// TIA Portal V19 export
FUNCTION_BLOCK "HMIGraphicControl"   // FB4, LAD
{ S7_Optimized_Access := 'TRUE' }
// stored: MemoryReserve 100, SetENOAutomatically false
   VAR_INPUT
      "Conveyor Speed" { ExternalAccessible := 'False'; ExternalVisible := 'False'; ExternalWritable := 'False'} : Real;   // m/min
      "Arm Speed" { ExternalAccessible := 'False'; ExternalVisible := 'False'; ExternalWritable := 'False'} : Real;   // m/min
      "Conveyor Max Speed" { ExternalAccessible := 'False'; ExternalVisible := 'False'; ExternalWritable := 'False'} : Real := 3000.0;
      "Arm Max Speed" { ExternalAccessible := 'False'; ExternalVisible := 'False'; ExternalWritable := 'False'} : Real := 32000.0;
      ConveyorMoving : Bool := true;
      ArmMoving : Bool := true;
      Reset : Bool;
   END_VAR
   VAR_OUTPUT
      Conveyor_On : Bool;
      Arm_On : Bool;
   END_VAR
   VAR_IN_OUT
      System_Enable : Bool;
      Graphic_Index { ExternalAccessible := 'False'; ExternalVisible := 'False'; ExternalWritable := 'False'} : Int;
      Box_Cnt : DInt;
      Pallet_Cnt : DInt;
   END_VAR
   VAR
      IEC_Timer_0_Instance { S7_SetPoint := 'True'} : IEC_TIMER;
      ConveyorTick : Bool;
      ConveyorTime : DInt;
      ConveyorTimeFactor : DInt := 100000;
      ArmTick : Bool;
      ArmTimeFactor : DInt := 100000;
      ArmTime : DInt;
      IEC_Timer_0_Instance_1 { S7_SetPoint := 'True'} : IEC_TIMER;
   END_VAR
   VAR_TEMP
      ConveyorScaled : Real;
      ConveyMotor : Bool;
      ArmScaled : Real;
   END_VAR
   VAR_TEMP   // added for the SCL form of the ladder/FBD networks
      _w1 : Bool;
   END_VAR
BEGIN

REGION Network 1
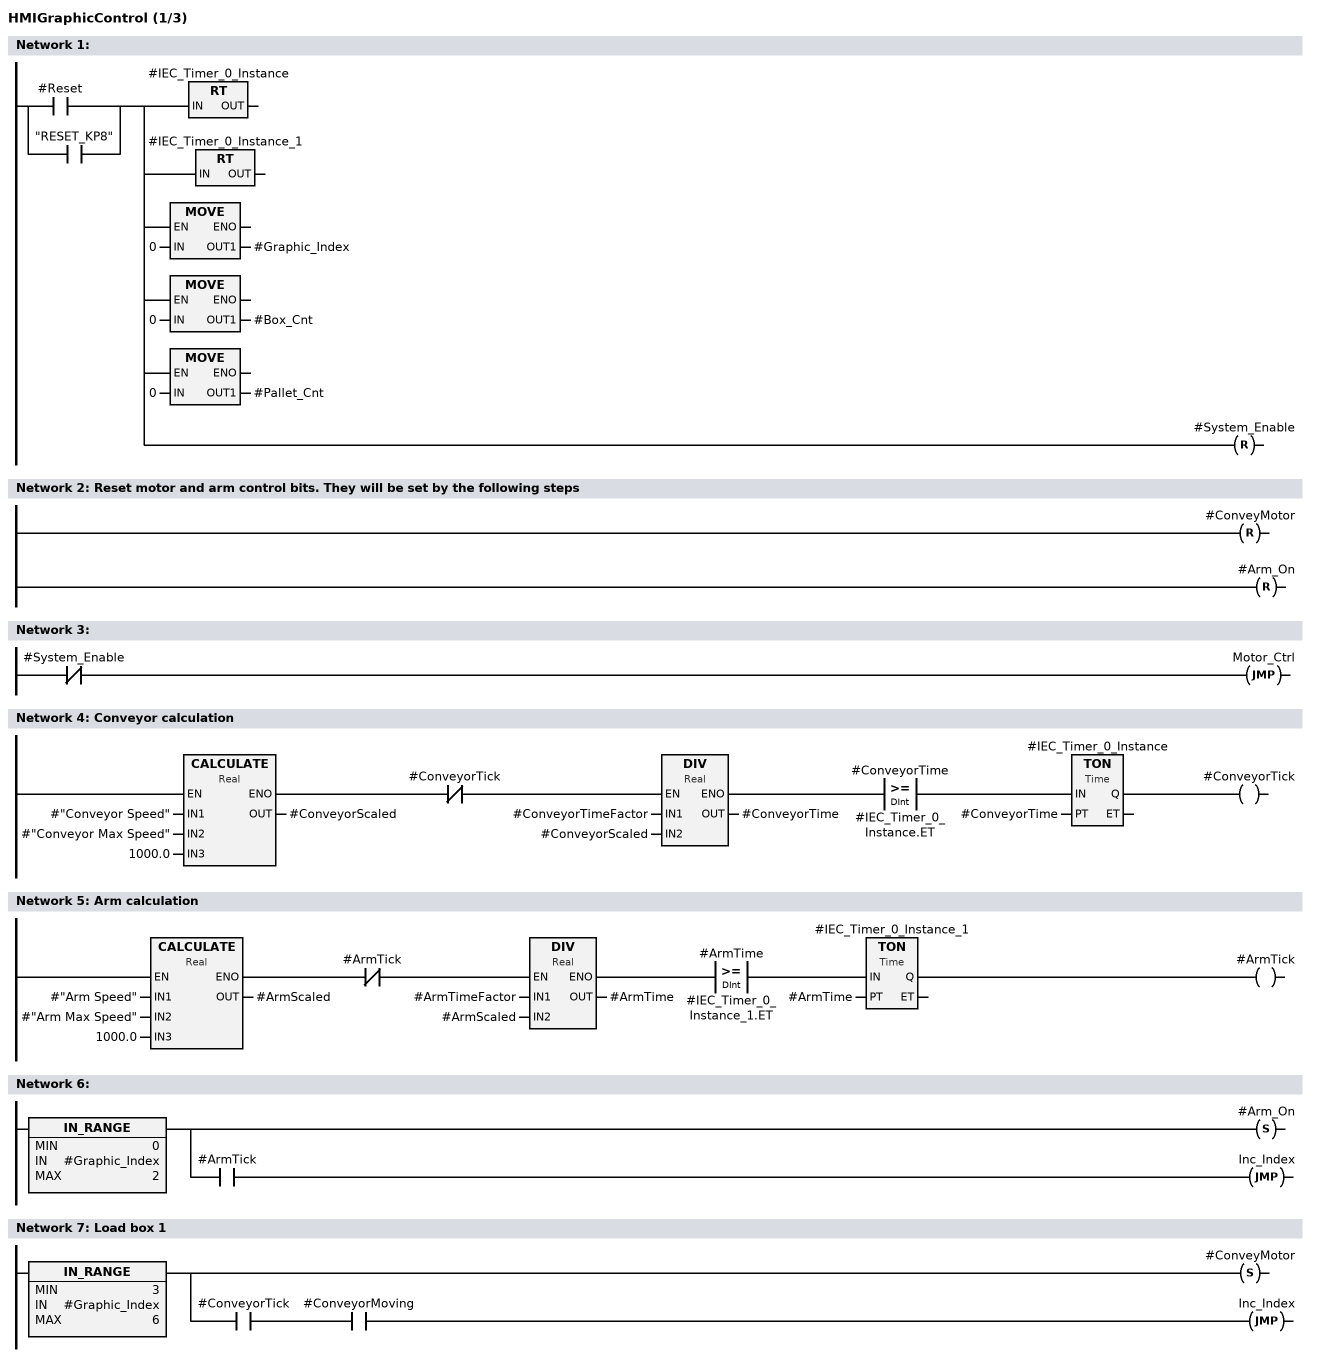
   RUNG wire#powerrail
      Contact( #Reset )
      wire#w1
      RT_Coil( #IEC_Timer_0_Instance )
   END_RUNG
   RUNG wire#powerrail
      Contact( "RESET_KP8" )
   END_RUNG wire#w1
   RUNG wire#w1
      RT_Coil( #IEC_Timer_0_Instance_1 )
   END_RUNG
   RUNG wire#w1
      Move(in := 0, out1 => #Graphic_Index)
   END_RUNG
   RUNG wire#w1
      Move(in := 0, out1 => #Box_Cnt)
   END_RUNG
   RUNG wire#w1
      Move(in := 0, out1 => #Pallet_Cnt)
   END_RUNG
   RUNG wire#w1
      R_Coil( #System_Enable )
   END_RUNG
   // the same network as SCL:
   #_w1 := #Reset OR "RESET_KP8";
   IF #_w1 THEN
       RESET_TIMER(#IEC_Timer_0_Instance);
       RESET_TIMER(#IEC_Timer_0_Instance_1);
       #Graphic_Index := 0;
       #Box_Cnt := 0;
       #Pallet_Cnt := 0;
       #System_Enable := FALSE;
   END_IF;
END_REGION

REGION Network 2: Reset motor and arm control bits. They will be set by the following steps
   RUNG wire#powerrail
      R_Coil( #ConveyMotor )
   END_RUNG
   RUNG wire#powerrail
      R_Coil( #Arm_On )
   END_RUNG
   // the same network as SCL:
   #ConveyMotor := FALSE;
   #Arm_On := FALSE;
END_REGION

REGION Network 3
   RUNG wire#powerrail
      I_Contact( #System_Enable )
      JumpCoil( Motor_Ctrl )
   END_RUNG
   // the same network as SCL:
   IF NOT #System_Enable THEN GOTO Motor_Ctrl; END_IF;
END_REGION

REGION Network 4: Conveyor calculation
   RUNG wire#powerrail
      { S7_Templates := "SrcType := Real"; S7_Expression := "IN1/IN2*IN3" } Calculate(in1 := #"Conveyor Speed", in2 := #"Conveyor Max Speed", in3 := 1000.0, out => #ConveyorScaled)
      I_Contact( #ConveyorTick )
      { S7_Templates := "SrcType := Real"; S7_GenerateENO := "TRUE" } Div(in1 := #ConveyorTimeFactor, in2 := #ConveyorScaled, out => #ConveyorTime)
      { S7_Templates := "SrcType := DInt" } GE_Contact(in1 := #ConveyorTime, in2 := #IEC_Timer_0_Instance.ET)
      { S7_Templates := "time_type := Time" } #IEC_Timer_0_Instance.TON(pt := #ConveyorTime, et =>)
      Coil( #ConveyorTick )
   END_RUNG
   // the same network as SCL:
   // ENO of a box is taken as its EN; it also drops when the box reports an error
   #ConveyorScaled := #"Conveyor Speed"/#"Conveyor Max Speed"*1000.0;
   IF NOT #ConveyorTick THEN #ConveyorTime := #ConveyorTimeFactor / #ConveyorScaled; END_IF;
   #IEC_Timer_0_Instance.TON(IN := NOT #ConveyorTick AND (#ConveyorTime >= #IEC_Timer_0_Instance.ET),
                           PT := #ConveyorTime);
   #ConveyorTick := #IEC_Timer_0_Instance.Q;
END_REGION

REGION Network 5: Arm calculation
   RUNG wire#powerrail
      { S7_Templates := "SrcType := Real"; S7_Expression := "IN1/IN2*IN3" } Calculate(in1 := #"Arm Speed", in2 := #"Arm Max Speed", in3 := 1000.0, out => #ArmScaled)
      I_Contact( #ArmTick )
      { S7_Templates := "SrcType := Real"; S7_GenerateENO := "TRUE" } Div(in1 := #ArmTimeFactor, in2 := #ArmScaled, out => #ArmTime)
      { S7_Templates := "SrcType := DInt" } GE_Contact(in1 := #ArmTime, in2 := #IEC_Timer_0_Instance_1.ET)
      { S7_Templates := "time_type := Time" } #IEC_Timer_0_Instance_1.TON(pt := #ArmTime, et =>)
      Coil( #ArmTick )
   END_RUNG
   // the same network as SCL:
   // ENO of a box is taken as its EN; it also drops when the box reports an error
   #ArmScaled := #"Arm Speed"/#"Arm Max Speed"*1000.0;
   IF NOT #ArmTick THEN #ArmTime := #ArmTimeFactor / #ArmScaled; END_IF;
   #IEC_Timer_0_Instance_1.TON(IN := NOT #ArmTick AND (#ArmTime >= #IEC_Timer_0_Instance_1.ET), PT := #ArmTime);
   #ArmTick := #IEC_Timer_0_Instance_1.Q;
END_REGION

REGION Network 6
   RUNG wire#powerrail
      { S7_Templates := "SrcType := Int" } InRange(min := 0, in := #Graphic_Index, max := 2)
      wire#w1
      S_Coil( #Arm_On )
   END_RUNG
   RUNG wire#w1
      Contact( #ArmTick )
      JumpCoil( Inc_Index )
   END_RUNG
   // the same network as SCL:
   #_w1 := (0 <= #Graphic_Index) AND (#Graphic_Index <= 2);
   IF #_w1 THEN #Arm_On := TRUE; END_IF;
   IF #_w1 AND #ArmTick THEN GOTO Inc_Index; END_IF;
END_REGION

REGION Network 7: Load box 1
   RUNG wire#powerrail
      { S7_Templates := "SrcType := Int" } InRange(min := 3, in := #Graphic_Index, max := 6)
      wire#w1
      S_Coil( #ConveyMotor )
   END_RUNG
   RUNG wire#w1
      Contact( #ConveyorTick )
      Contact( #ConveyorMoving )
      JumpCoil( Inc_Index )
   END_RUNG
   // the same network as SCL:
   #_w1 := (3 <= #Graphic_Index) AND (#Graphic_Index <= 6);
   IF #_w1 THEN #ConveyMotor := TRUE; END_IF;
   IF #_w1 AND #ConveyorTick AND #ConveyorMoving THEN GOTO Inc_Index; END_IF;
END_REGION

REGION Network 8
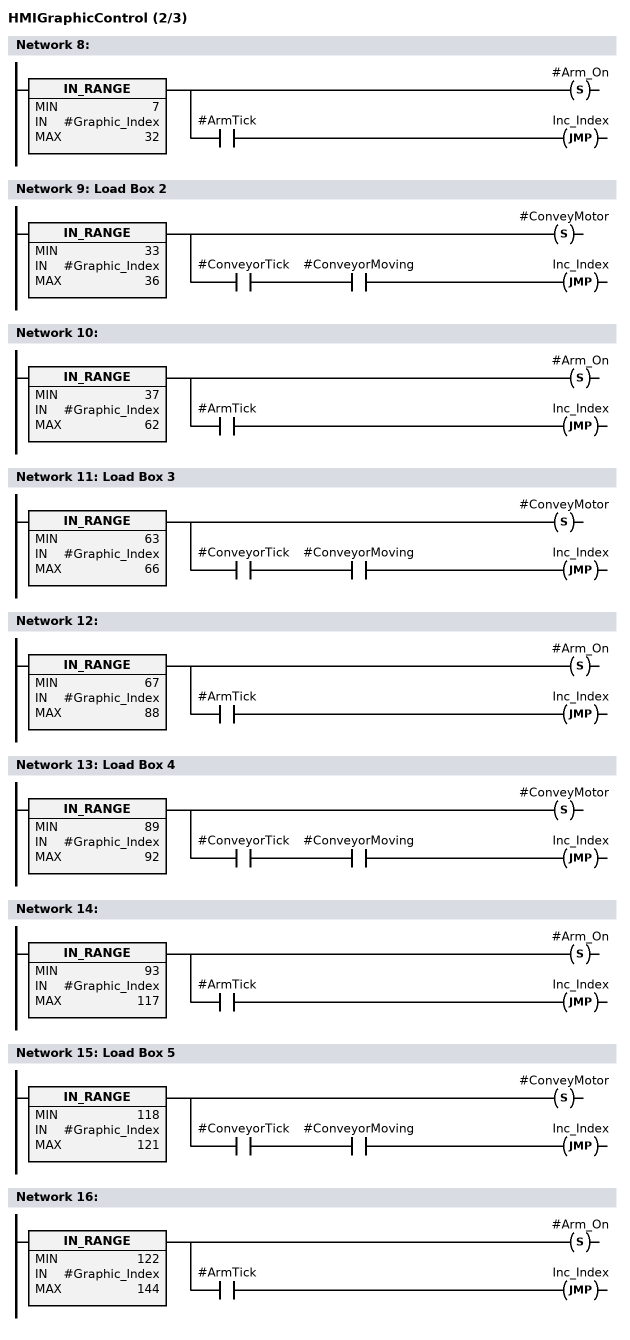
   RUNG wire#powerrail
      { S7_Templates := "SrcType := Int" } InRange(min := 7, in := #Graphic_Index, max := 32)
      wire#w1
      S_Coil( #Arm_On )
   END_RUNG
   RUNG wire#w1
      Contact( #ArmTick )
      JumpCoil( Inc_Index )
   END_RUNG
   // the same network as SCL:
   #_w1 := (7 <= #Graphic_Index) AND (#Graphic_Index <= 32);
   IF #_w1 THEN #Arm_On := TRUE; END_IF;
   IF #_w1 AND #ArmTick THEN GOTO Inc_Index; END_IF;
END_REGION

REGION Network 9: Load Box 2
   RUNG wire#powerrail
      { S7_Templates := "SrcType := Int" } InRange(min := 33, in := #Graphic_Index, max := 36)
      wire#w1
      S_Coil( #ConveyMotor )
   END_RUNG
   RUNG wire#w1
      Contact( #ConveyorTick )
      Contact( #ConveyorMoving )
      JumpCoil( Inc_Index )
   END_RUNG
   // the same network as SCL:
   #_w1 := (33 <= #Graphic_Index) AND (#Graphic_Index <= 36);
   IF #_w1 THEN #ConveyMotor := TRUE; END_IF;
   IF #_w1 AND #ConveyorTick AND #ConveyorMoving THEN GOTO Inc_Index; END_IF;
END_REGION

REGION Network 10
   RUNG wire#powerrail
      { S7_Templates := "SrcType := Int" } InRange(min := 37, in := #Graphic_Index, max := 62)
      wire#w1
      S_Coil( #Arm_On )
   END_RUNG
   RUNG wire#w1
      Contact( #ArmTick )
      JumpCoil( Inc_Index )
   END_RUNG
   // the same network as SCL:
   #_w1 := (37 <= #Graphic_Index) AND (#Graphic_Index <= 62);
   IF #_w1 THEN #Arm_On := TRUE; END_IF;
   IF #_w1 AND #ArmTick THEN GOTO Inc_Index; END_IF;
END_REGION

REGION Network 11: Load Box 3
   RUNG wire#powerrail
      { S7_Templates := "SrcType := Int" } InRange(min := 63, in := #Graphic_Index, max := 66)
      wire#w1
      S_Coil( #ConveyMotor )
   END_RUNG
   RUNG wire#w1
      Contact( #ConveyorTick )
      Contact( #ConveyorMoving )
      JumpCoil( Inc_Index )
   END_RUNG
   // the same network as SCL:
   #_w1 := (63 <= #Graphic_Index) AND (#Graphic_Index <= 66);
   IF #_w1 THEN #ConveyMotor := TRUE; END_IF;
   IF #_w1 AND #ConveyorTick AND #ConveyorMoving THEN GOTO Inc_Index; END_IF;
END_REGION

REGION Network 12
   RUNG wire#powerrail
      { S7_Templates := "SrcType := Int" } InRange(min := 67, in := #Graphic_Index, max := 88)
      wire#w1
      S_Coil( #Arm_On )
   END_RUNG
   RUNG wire#w1
      Contact( #ArmTick )
      JumpCoil( Inc_Index )
   END_RUNG
   // the same network as SCL:
   #_w1 := (67 <= #Graphic_Index) AND (#Graphic_Index <= 88);
   IF #_w1 THEN #Arm_On := TRUE; END_IF;
   IF #_w1 AND #ArmTick THEN GOTO Inc_Index; END_IF;
END_REGION

REGION Network 13: Load Box 4
   RUNG wire#powerrail
      { S7_Templates := "SrcType := Int" } InRange(min := 89, in := #Graphic_Index, max := 92)
      wire#w1
      S_Coil( #ConveyMotor )
   END_RUNG
   RUNG wire#w1
      Contact( #ConveyorTick )
      Contact( #ConveyorMoving )
      JumpCoil( Inc_Index )
   END_RUNG
   // the same network as SCL:
   #_w1 := (89 <= #Graphic_Index) AND (#Graphic_Index <= 92);
   IF #_w1 THEN #ConveyMotor := TRUE; END_IF;
   IF #_w1 AND #ConveyorTick AND #ConveyorMoving THEN GOTO Inc_Index; END_IF;
END_REGION

REGION Network 14
   RUNG wire#powerrail
      { S7_Templates := "SrcType := Int" } InRange(min := 93, in := #Graphic_Index, max := 117)
      wire#w1
      S_Coil( #Arm_On )
   END_RUNG
   RUNG wire#w1
      Contact( #ArmTick )
      JumpCoil( Inc_Index )
   END_RUNG
   // the same network as SCL:
   #_w1 := (93 <= #Graphic_Index) AND (#Graphic_Index <= 117);
   IF #_w1 THEN #Arm_On := TRUE; END_IF;
   IF #_w1 AND #ArmTick THEN GOTO Inc_Index; END_IF;
END_REGION

REGION Network 15: Load Box 5
   RUNG wire#powerrail
      { S7_Templates := "SrcType := Int" } InRange(min := 118, in := #Graphic_Index, max := 121)
      wire#w1
      S_Coil( #ConveyMotor )
   END_RUNG
   RUNG wire#w1
      Contact( #ConveyorTick )
      Contact( #ConveyorMoving )
      JumpCoil( Inc_Index )
   END_RUNG
   // the same network as SCL:
   #_w1 := (118 <= #Graphic_Index) AND (#Graphic_Index <= 121);
   IF #_w1 THEN #ConveyMotor := TRUE; END_IF;
   IF #_w1 AND #ConveyorTick AND #ConveyorMoving THEN GOTO Inc_Index; END_IF;
END_REGION

REGION Network 16
   RUNG wire#powerrail
      { S7_Templates := "SrcType := Int" } InRange(min := 122, in := #Graphic_Index, max := 144)
      wire#w1
      S_Coil( #Arm_On )
   END_RUNG
   RUNG wire#w1
      Contact( #ArmTick )
      JumpCoil( Inc_Index )
   END_RUNG
   // the same network as SCL:
   #_w1 := (122 <= #Graphic_Index) AND (#Graphic_Index <= 144);
   IF #_w1 THEN #Arm_On := TRUE; END_IF;
   IF #_w1 AND #ArmTick THEN GOTO Inc_Index; END_IF;
END_REGION

REGION Network 17: Load Box 6
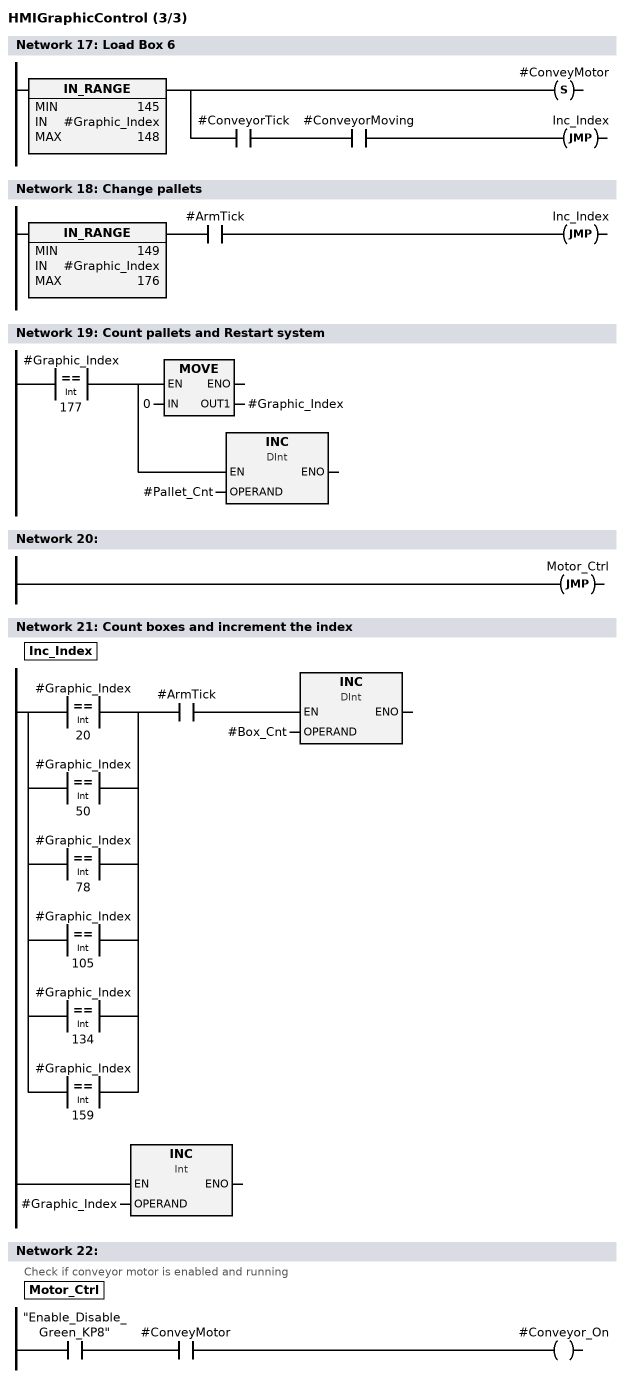
   RUNG wire#powerrail
      { S7_Templates := "SrcType := Int" } InRange(min := 145, in := #Graphic_Index, max := 148)
      wire#w1
      S_Coil( #ConveyMotor )
   END_RUNG
   RUNG wire#w1
      Contact( #ConveyorTick )
      Contact( #ConveyorMoving )
      JumpCoil( Inc_Index )
   END_RUNG
   // the same network as SCL:
   #_w1 := (145 <= #Graphic_Index) AND (#Graphic_Index <= 148);
   IF #_w1 THEN #ConveyMotor := TRUE; END_IF;
   IF #_w1 AND #ConveyorTick AND #ConveyorMoving THEN GOTO Inc_Index; END_IF;
END_REGION

REGION Network 18: Change pallets
   RUNG wire#powerrail
      { S7_Templates := "SrcType := Int" } InRange(min := 149, in := #Graphic_Index, max := 176)
      Contact( #ArmTick )
      JumpCoil( Inc_Index )
   END_RUNG
   // the same network as SCL:
   IF (149 <= #Graphic_Index) AND (#Graphic_Index <= 176) AND #ArmTick THEN GOTO Inc_Index; END_IF;
END_REGION

REGION Network 19: Count pallets and Restart system
   RUNG wire#powerrail
      { S7_Templates := "SrcType := Int" } EQ_Contact(in1 := #Graphic_Index, in2 := 177)
      wire#w1
      Move(in := 0, out1 => #Graphic_Index)
   END_RUNG
   RUNG wire#w1
      { S7_Templates := "DestType := DInt" } Inc( #Pallet_Cnt )
   END_RUNG
   // the same network as SCL:
   #_w1 := #Graphic_Index = 177;
   IF #_w1 THEN
       #Graphic_Index := 0;
       #Pallet_Cnt := #Pallet_Cnt + 1;
   END_IF;
END_REGION

REGION Network 20
   RUNG wire#powerrail
      JumpCoil( Motor_Ctrl )
   END_RUNG
   // the same network as SCL:
   GOTO Motor_Ctrl;
END_REGION

REGION Network 21: Count boxes and increment the index
   Label( Inc_Index )
   RUNG wire#powerrail
      { S7_Templates := "SrcType := Int" } EQ_Contact(in1 := #Graphic_Index, in2 := 20)
      wire#w1
      Contact( #ArmTick )
      { S7_Templates := "DestType := DInt" } Inc( #Box_Cnt )
   END_RUNG
   RUNG wire#powerrail
      { S7_Templates := "SrcType := Int" } EQ_Contact(in1 := #Graphic_Index, in2 := 50)
   END_RUNG wire#w1
   RUNG wire#powerrail
      { S7_Templates := "SrcType := Int" } EQ_Contact(in1 := #Graphic_Index, in2 := 78)
   END_RUNG wire#w1
   RUNG wire#powerrail
      { S7_Templates := "SrcType := Int" } EQ_Contact(in1 := #Graphic_Index, in2 := 105)
   END_RUNG wire#w1
   RUNG wire#powerrail
      { S7_Templates := "SrcType := Int" } EQ_Contact(in1 := #Graphic_Index, in2 := 134)
   END_RUNG wire#w1
   RUNG wire#powerrail
      { S7_Templates := "SrcType := Int" } EQ_Contact(in1 := #Graphic_Index, in2 := 159)
   END_RUNG wire#w1
   RUNG wire#powerrail
      { S7_Templates := "DestType := Int" } Inc( #Graphic_Index )
   END_RUNG
   // the same network as SCL:
   Inc_Index:
   IF ((#Graphic_Index = 20) OR (#Graphic_Index = 50) OR (#Graphic_Index = 78) OR (#Graphic_Index = 105) OR (#Graphic_Index = 134) OR (#Graphic_Index = 159)) AND #ArmTick THEN
       #Box_Cnt := #Box_Cnt + 1;
   END_IF;
   #Graphic_Index := #Graphic_Index + 1;
END_REGION

REGION Network 22
   // Check if conveyor motor is enabled and running
   Label( Motor_Ctrl )
   RUNG wire#powerrail
      Contact( "Enable_Disable_Green_KP8" )
      Contact( #ConveyMotor )
      Coil( #Conveyor_On )
   END_RUNG
   // the same network as SCL:
   Motor_Ctrl:
   #Conveyor_On := "Enable_Disable_Green_KP8" AND #ConveyMotor;
END_REGION
END_FUNCTION_BLOCK
